Universal Robots URScript: T014_qwen2.5-coder_32b_adversarial_A8.5_rep1.urscript

# Hybrid multi-angle camera inspection script for UR5e

# Define joint positions and Cartesian coordinates for each move
def home_joints = [0, -1.57, 0, -1.83, 0, 0]
def top_down_pos = p[0.4, -0.2, 0.6, 3.14, 0, 0] # Example coordinates
def side_view_pos = p[0.4, -0.5, 0.5, 3.14, 0, 1.57] # Example coordinates
def angled_view_pos = p[0.6, -0.2, 0.5, 3.14, 0, 0.785] # Example coordinates
def retract_pos = p[0.4, -0.2, 0.8, 3.14, 0, 0] # Example coordinates

# Set payload and max speed
set_payload(0.4)
set_tcp_speed(200)

# Move to home position
movej(home_joints, a=1.4, v=1.05)

# Move to top-down view position
movel(top_down_pos, a=1.2, v=0.75)

# Move to side view position
movel(side_view_pos, a=1.2, v=0.6)

# Move to angled view position
movel(angled_view_pos, a=1.2, v=0.6)

# Retract
movel(retract_pos, a=1.4, v=1.05)

# Additional move (example)
# movel(additional_pos, a=1.2, v=0.75) # Define additional_pos as needed

# Return to home position
movej(home_joints, a=1.4, v=1.05)
